FUNCTION_BLOCK EL5152
VAR
	_io : EL5152_Data;
	{attribute addProperty Name "WcState"}
	_wcState : WcStateInputToggle;
	{attribute addProperty Name "Info data"}
	_infoData : InfoDataAdsDC;
END_VAR

PROPERTY IO : REFERENCE TO EL5152_Data
GET
IO REF= _io;
END_GET
END_PROPERTY

PROPERTY WcState : REFERENCE TO WcStateInputToggle
GET
WcState REF= _wcState;
END_GET
END_PROPERTY

END_FUNCTION_BLOCK

(* stored: Version 1.1.0.1, ProductVersion 3.1.4024.9
   POU EL5152: Id {c9a01d29-0b42-0425-21dc-f2b25e39b10d}, SpecialFunc None
   Property IO: Id {7fd0ec34-47a8-0fa2-24dc-c3efc20bdeed}
   Get Get: Id {507d2c81-d7af-04d9-2774-c2ced2c5f55a}
   Property WcState: Id {de0c24b9-496b-0f9b-1b75-ec578977799b}
   Get Get: Id {8d00daa4-3961-061f-0cea-7e5e2d9fcfa6} *)
